// TIA Portal V16 export
// export: Created 2022-01-20T19:04:41.3515111Z, ExportSetting WithDefaults, DisplayName Totally Integrated Automation Portal, DisplayVersion V16, DisplayName TIA Portal Version Control Interface, DisplayVersion V16, DisplayName TIA Portal Openness, DisplayVersion V16, DisplayName STEP 7 Professional, DisplayVersion V16, DisplayName STEP 7 Safety, DisplayVersion V16, DisplayName WinCC Advanced, DisplayVersion V16
ORGANIZATION_BLOCK "Main"   // OB1, LAD, ProgramCycle
TITLE = "Main Program Sweep (Cycle)"
{ S7_Optimized_Access := 'TRUE' }
VERSION : 0.1
// stored: AutoNumber true, IsIECCheckEnabled false, SetENOAutomatically false
   VAR_INPUT
      Initial_Call : Bool;   // Initial call of this OB
      Remanence : Bool;   // =True, if remanent data are available
   END_VAR
   VAR_TEMP
      suma : Int;
   END_VAR
BEGIN

REGION Network 1
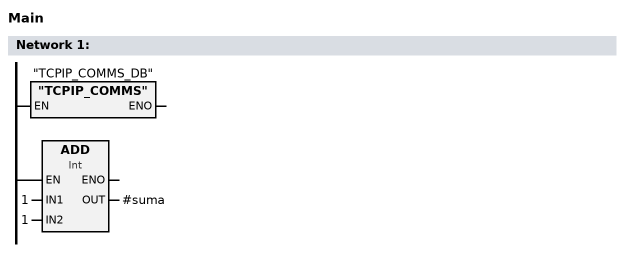
   RUNG wire#powerrail
      "TCPIP_COMMS_DB"()
   END_RUNG
   RUNG wire#powerrail
      { S7_Templates := "SrcType := Int" } Add(in1 := 1, in2 := 1, out => #suma)
   END_RUNG
   // the same network as SCL:
   "TCPIP_COMMS_DB"();   // "TCPIP_COMMS"
   #suma := 1 + 1;
END_REGION
END_ORGANIZATION_BLOCK
